// TIA Portal V20 export
FUNCTION "LER_VisionCommand" : Void   // FC106, LAD
// stored: Access Published, SetENOAutomatically false
   VAR_INPUT
      enable : Bool;
   END_VAR
   VAR_IN_OUT
      Command : USInt;
      Vison : "LER_typeVisionControlNode";
   END_VAR
   VAR CONSTANT
      CommandReset : USInt;
      CommandStepStart : USInt := 1;
   END_VAR
BEGIN

REGION Network 2
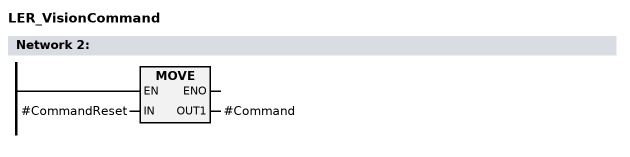
   RUNG wire#powerrail
      Move(in := #CommandReset, out1 => #Command)
   END_RUNG
   // the same network as SCL:
   #Command := #CommandReset;
END_REGION
END_FUNCTION
